(* PLC project Tc3_EventLogger.ResetToDefault Demo, tc3-libraries-kb TwinCAT 3.1 *)
(* stored: creationDateTime 2026-05-11T01:00:00, modificationDateTime 2026-05-11T01:00:00 *)

PROGRAM P_Demo_ResetToDefault
  VAR
    fbSrc : FB_TcSourceInfo;  (* 源信息实例 *)
    bDoReset : BOOL := FALSE;  (* 上升沿触发 *)
    bDoResetPrev : BOOL;  (* 边沿检测 *)
    hr : HRESULT;  (* 返回值监视 *)
  END_VAR

// =============================================================================
// 场景：测试结束后还原 SourceInfo 到默认
// 价值：一次调用还原
// 验证：登录后调用 ResetToDefault 后 fbSrc 字段回到默认（SourceName = PLC 符号路径）
// 验证步骤：
//   1. 右键 PLC 项目 → Import PLCopenXML → 选本文件
//   2. 引用 Tc3_EventLogger（System → References → Add library）
//   3. 编译 → 登录 → 运行；按 verify 注释里给出的在线写值操作
// =============================================================================

IF bDoReset AND NOT bDoResetPrev THEN
    hr := fbSrc.ResetToDefault();
END_IF;
bDoResetPrev := bDoReset;
END_PROGRAM
